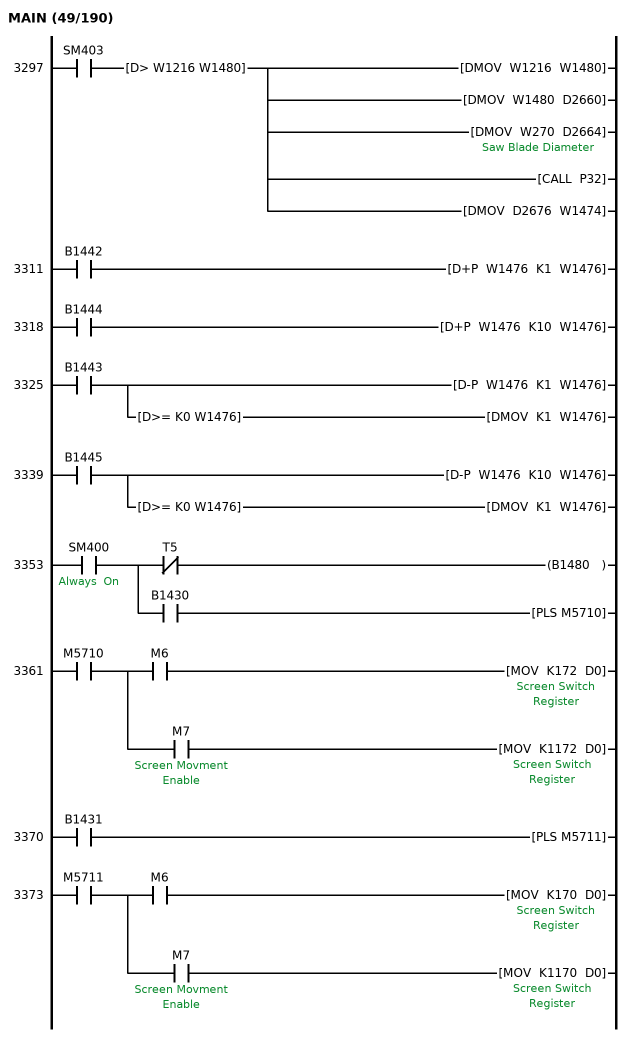
[picture p48: ladder of MAIN, rungs at steps 3297 to 3373]
3297  LD      SM403
      ANDD>   W1216 W1480
      DMOV    W1216 W1480
      DMOV    W1480 D2660
      DMOV    W270 D2664
      CALL    P32
      DMOV    D2676 W1474
3311  LD      B1442
      D+P     W1476 K1 W1476
3318  LD      B1444
      D+P     W1476 K10 W1476
3325  LD      B1443
      D-P     W1476 K1 W1476
      ANDD>=  K0 W1476
      DMOV    K1 W1476
3339  LD      B1445
      D-P     W1476 K10 W1476
      ANDD>=  K0 W1476
      DMOV    K1 W1476
3353  LD      SM400  ; Always  On
      MPS
      ANI     T5
      OUT     B1480
      MPP
      AND     B1430
      PLS     M5710
3361  LD      M5710
      MPS
      AND     M6
      MOV     K172 D0
      MPP
      AND     M7  ; Screen Movment Enable
      MOV     K1172 D0
3370  LD      B1431
      PLS     M5711
3373  LD      M5711
      MPS
      AND     M6
      MOV     K170 D0
      MPP
      AND     M7  ; Screen Movment Enable
      MOV     K1170 D0
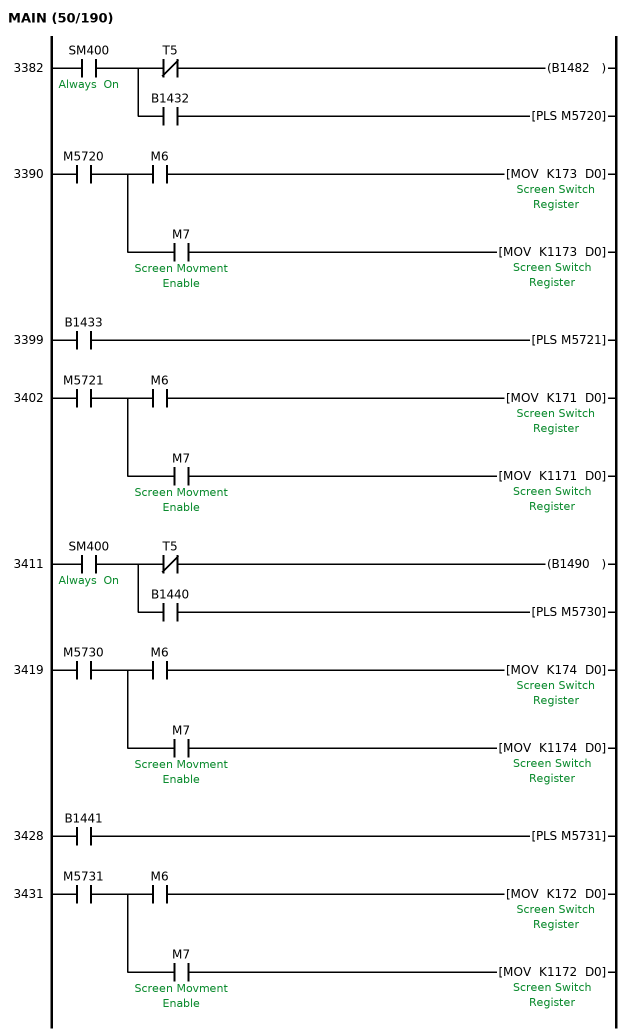
3382  LD      SM400  ; Always  On
      MPS
      ANI     T5
      OUT     B1482
      MPP
      AND     B1432
      PLS     M5720
3390  LD      M5720
      MPS
      AND     M6
      MOV     K173 D0
      MPP
      AND     M7  ; Screen Movment Enable
      MOV     K1173 D0
3399  LD      B1433
      PLS     M5721
3402  LD      M5721
      MPS
      AND     M6
      MOV     K171 D0
      MPP
      AND     M7  ; Screen Movment Enable
      MOV     K1171 D0
3411  LD      SM400  ; Always  On
      MPS
      ANI     T5
      OUT     B1490
      MPP
      AND     B1440
      PLS     M5730
3419  LD      M5730
      MPS
      AND     M6
      MOV     K174 D0
      MPP
      AND     M7  ; Screen Movment Enable
      MOV     K1174 D0
3428  LD      B1441
      PLS     M5731
3431  LD      M5731
      MPS
      AND     M6
      MOV     K172 D0
      MPP
      AND     M7  ; Screen Movment Enable
      MOV     K1172 D0
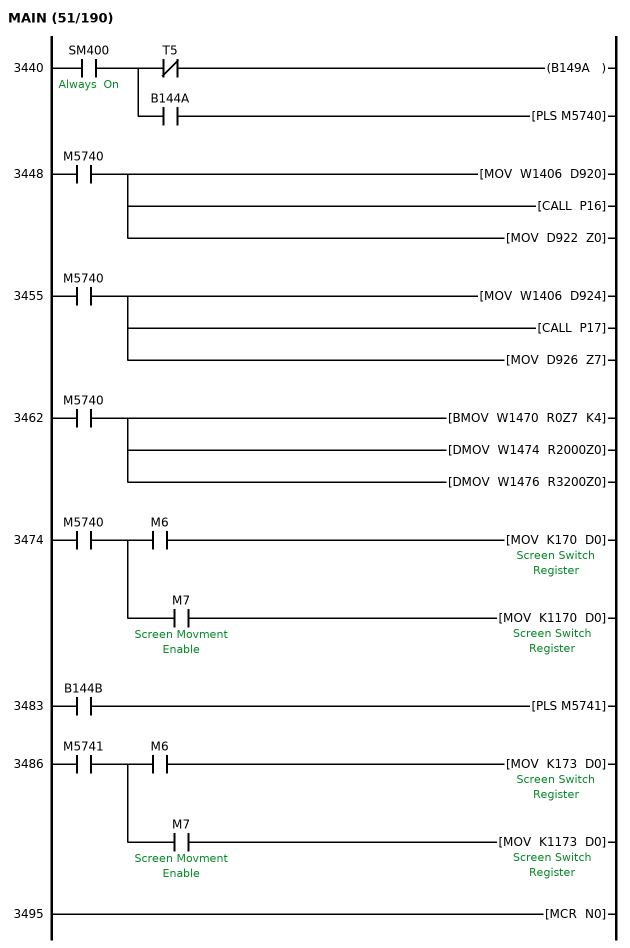
3440  LD      SM400  ; Always  On
      MPS
      ANI     T5
      OUT     B149A
      MPP
      AND     B144A
      PLS     M5740
3448  LD      M5740
      MOV     W1406 D920
      CALL    P16
      MOV     D922 Z0
3455  LD      M5740
      MOV     W1406 D924
      CALL    P17
      MOV     D926 Z7
3462  LD      M5740
      BMOV    W1470 R0Z7 K4
      DMOV    W1474 R2000Z0
      DMOV    W1476 R3200Z0
3474  LD      M5740
      MPS
      AND     M6
      MOV     K170 D0
      MPP
      AND     M7  ; Screen Movment Enable
      MOV     K1170 D0
3483  LD      B144B
      PLS     M5741
3486  LD      M5741
      MPS
      AND     M6
      MOV     K173 D0
      MPP
      AND     M7  ; Screen Movment Enable
      MOV     K1173 D0
3495  MCR     N0
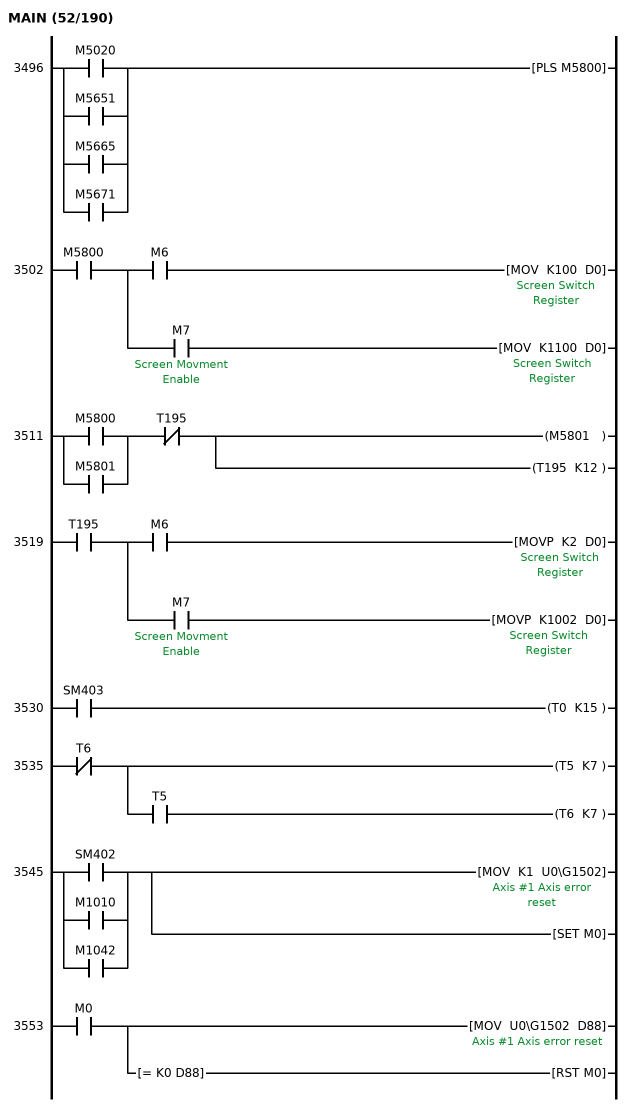
3496  LD      M5020
      OR      M5651
      OR      M5665
      OR      M5671
      PLS     M5800
3502  LD      M5800
      MPS
      AND     M6
      MOV     K100 D0
      MPP
      AND     M7  ; Screen Movment Enable
      MOV     K1100 D0
3511  LD      M5800
      OR      M5801
      ANI     T195
      OUT     M5801
      OUT     T195 K12
3519  LD      T195
      MPS
      AND     M6
      MOVP    K2 D0
      MPP
      AND     M7  ; Screen Movment Enable
      MOVP    K1002 D0
3530  LD      SM403
      OUT     T0 K15
3535  LDI     T6
      OUT     T5 K7
      AND     T5
      OUT     T6 K7
3545  LD      SM402
      OR      M1010
      OR      M1042
      MOV     K1 U0\G1502  ; Axis #1 Axis error reset
      SET     M0
3553  LD      M0
      MOV     U0\G1502 D88
      AND=    K0 D88
      RST     M0
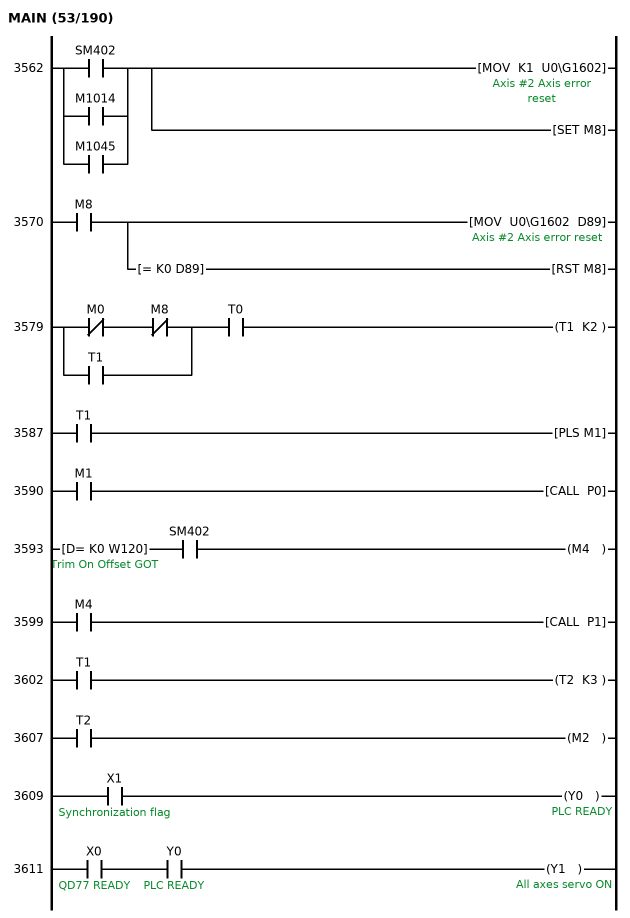
3562  LD      SM402
      OR      M1014
      OR      M1045
      MOV     K1 U0\G1602  ; Axis #2 Axis error reset
      SET     M8
3570  LD      M8
      MOV     U0\G1602 D89
      AND=    K0 D89
      RST     M8
3579  LDI     M0
      ANI     M8
      OR      T1
      AND     T0
      OUT     T1 K2
3587  LD      T1
      PLS     M1
3590  LD      M1
      CALL    P0
3593  LDD=    K0 W120  ; Trim On Offset GOT
      AND     SM402
      OUT     M4
3599  LD      M4
      CALL    P1
3602  LD      T1
      OUT     T2 K3
3607  LD      T2
      OUT     M2
3609  LD      X1  ; Synchronization flag
      OUT     Y0  ; PLC READY
3611  LD      X0  ; QD77 READY
      AND     Y0  ; PLC READY
      OUT     Y1  ; All axes servo ON
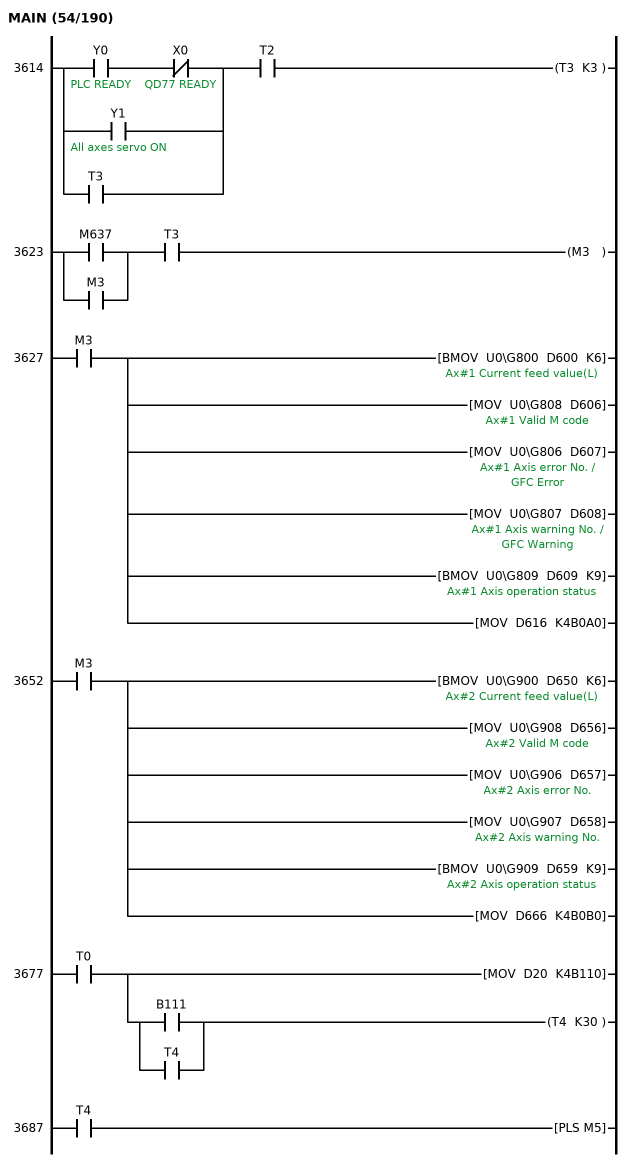
3614  LD      Y0  ; PLC READY
      ANI     X0  ; QD77 READY
      OR      Y1  ; All axes servo ON
      OR      T3
      AND     T2
      OUT     T3 K3
3623  LD      M637
      OR      M3
      AND     T3
      OUT     M3
3627  LD      M3
      BMOV    U0\G800 D600 K6  ; Ax#1 Current feed value(L)
      MOV     U0\G808 D606  ; Ax#1 Valid M code
      MOV     U0\G806 D607  ; Ax#1 Axis error No. / GFC Error
      MOV     U0\G807 D608  ; Ax#1 Axis warning No. / GFC Warning
      BMOV    U0\G809 D609 K9  ; Ax#1 Axis operation status
      MOV     D616 K4B0A0
3652  LD      M3
      BMOV    U0\G900 D650 K6  ; Ax#2 Current feed value(L)
      MOV     U0\G908 D656  ; Ax#2 Valid M code
      MOV     U0\G906 D657  ; Ax#2 Axis error No.
      MOV     U0\G907 D658  ; Ax#2 Axis warning No.
      BMOV    U0\G909 D659 K9  ; Ax#2 Axis operation status
      MOV     D666 K4B0B0
3677  LD      T0
      MOV     D20 K4B110
      LD      B111
      OR      T4
      ANB
      OUT     T4 K30
3687  LD      T4
      PLS     M5
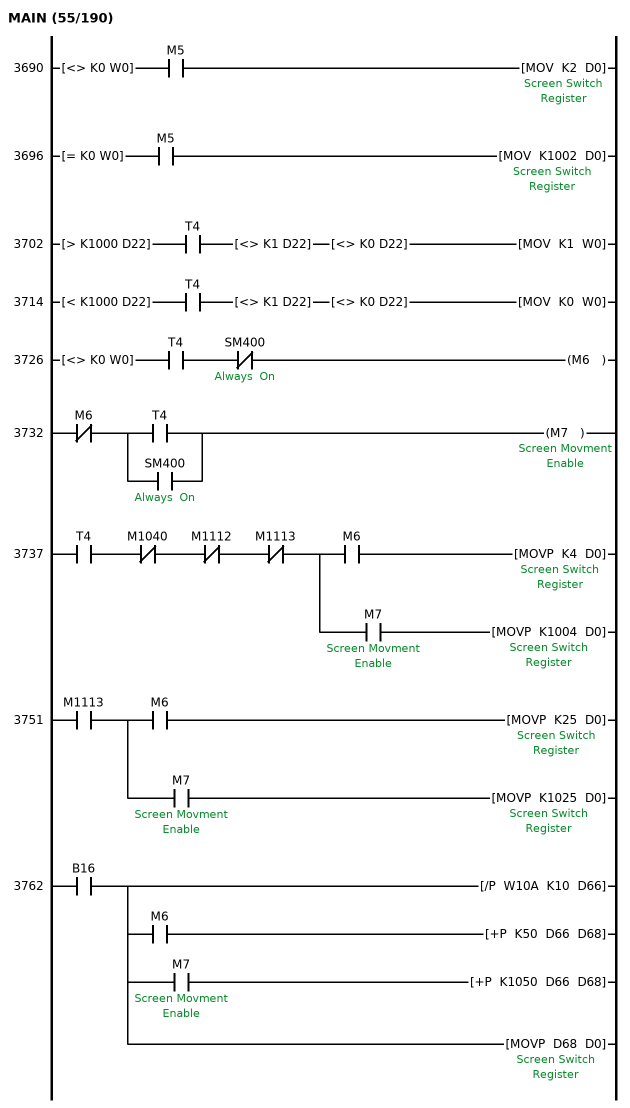
3690  LD<>    K0 W0
      AND     M5
      MOV     K2 D0
3696  LD=     K0 W0
      AND     M5
      MOV     K1002 D0
3702  LD>     K1000 D22
      AND     T4
      AND<>   K1 D22
      AND<>   K0 D22
      MOV     K1 W0
3714  LD<     K1000 D22
      AND     T4
      AND<>   K1 D22
      AND<>   K0 D22
      MOV     K0 W0
3726  LD<>    K0 W0
      AND     T4
      ANI     SM400  ; Always  On
      OUT     M6
3732  LDI     M6
      LD      T4
      OR      SM400  ; Always  On
      ANB
      OUT     M7  ; Screen Movment Enable
3737  LD      T4
      ANI     M1040
      ANI     M1112
      ANI     M1113
      MPS
      AND     M6
      MOVP    K4 D0
      MPP
      AND     M7  ; Screen Movment Enable
      MOVP    K1004 D0
3751  LD      M1113
      MPS
      AND     M6
      MOVP    K25 D0
      MPP
      AND     M7  ; Screen Movment Enable
      MOVP    K1025 D0
3762  LD      B16
      /P      W10A K10 D66
      MPS
      AND     M6
      +P      K50 D66 D68
      MRD
      AND     M7  ; Screen Movment Enable
      +P      K1050 D66 D68
      MPP
      MOVP    D68 D0
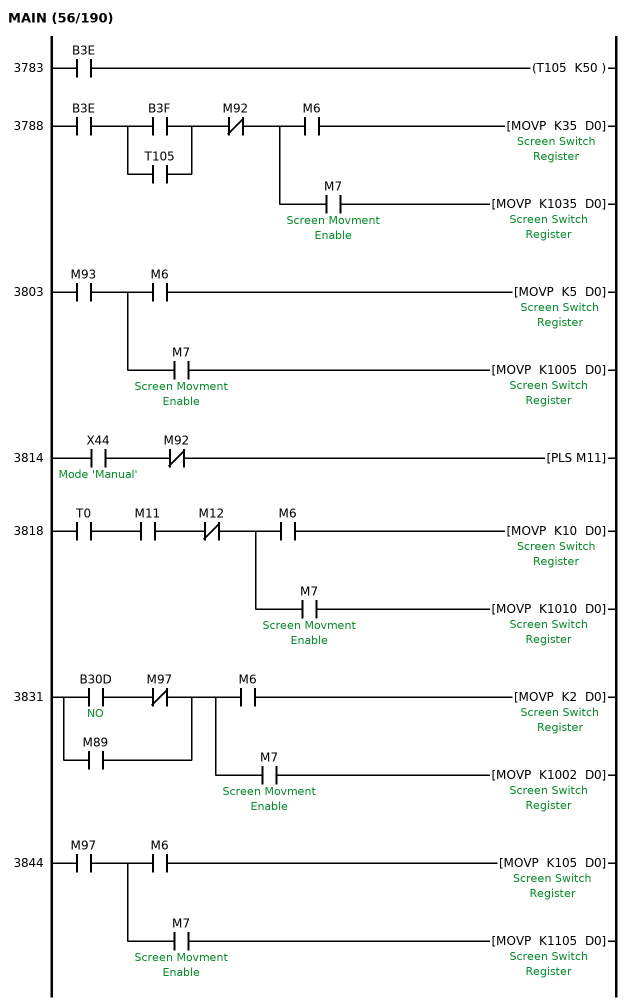
3783  LD      B3E
      OUT     T105 K50
3788  LD      B3E
      LD      B3F
      OR      T105
      ANB
      ANI     M92
      MPS
      AND     M6
      MOVP    K35 D0
      MPP
      AND     M7  ; Screen Movment Enable
      MOVP    K1035 D0
3803  LD      M93
      MPS
      AND     M6
      MOVP    K5 D0
      MPP
      AND     M7  ; Screen Movment Enable
      MOVP    K1005 D0
3814  LD      X44  ; Mode 'Manual'
      ANI     M92
      PLS     M11
3818  LD      T0
      AND     M11
      ANI     M12
      MPS
      AND     M6
      MOVP    K10 D0
      MPP
      AND     M7  ; Screen Movment Enable
      MOVP    K1010 D0
3831  LD      B30D  ; NO
      ANI     M97
      OR      M89
      MPS
      AND     M6
      MOVP    K2 D0
      MPP
      AND     M7  ; Screen Movment Enable
      MOVP    K1002 D0
3844  LD      M97
      MPS
      AND     M6
      MOVP    K105 D0
      MPP
      AND     M7  ; Screen Movment Enable
      MOVP    K1105 D0
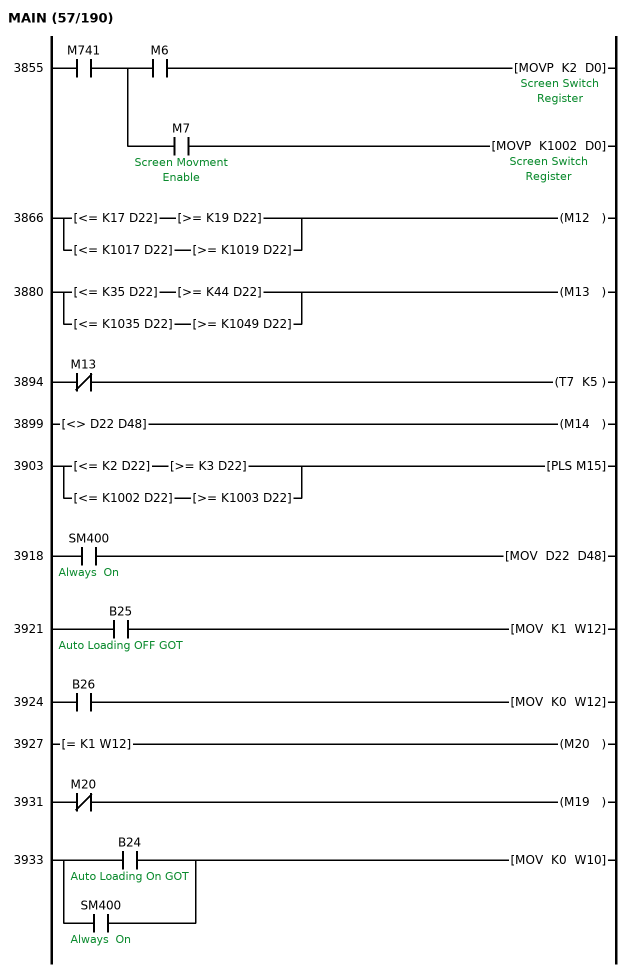
3855  LD      M741
      MPS
      AND     M6
      MOVP    K2 D0
      MPP
      AND     M7  ; Screen Movment Enable
      MOVP    K1002 D0
3866  LD<=    K17 D22
      AND>=   K19 D22
      LD<=    K1017 D22
      AND>=   K1019 D22
      ORB
      OUT     M12
3880  LD<=    K35 D22
      AND>=   K44 D22
      LD<=    K1035 D22
      AND>=   K1049 D22
      ORB
      OUT     M13
3894  LDI     M13
      OUT     T7 K5
3899  LD<>    D22 D48
      OUT     M14
3903  LD<=    K2 D22
      AND>=   K3 D22
      LD<=    K1002 D22
      AND>=   K1003 D22
      ORB
      PLS     M15
3918  LD      SM400  ; Always  On
      MOV     D22 D48
3921  LD      B25  ; Auto Loading OFF GOT
      MOV     K1 W12
3924  LD      B26
      MOV     K0 W12
3927  LD=     K1 W12
      OUT     M20
3931  LDI     M20
      OUT     M19
3933  LD      B24  ; Auto Loading On GOT
      OR      SM400  ; Always  On
      MOV     K0 W10
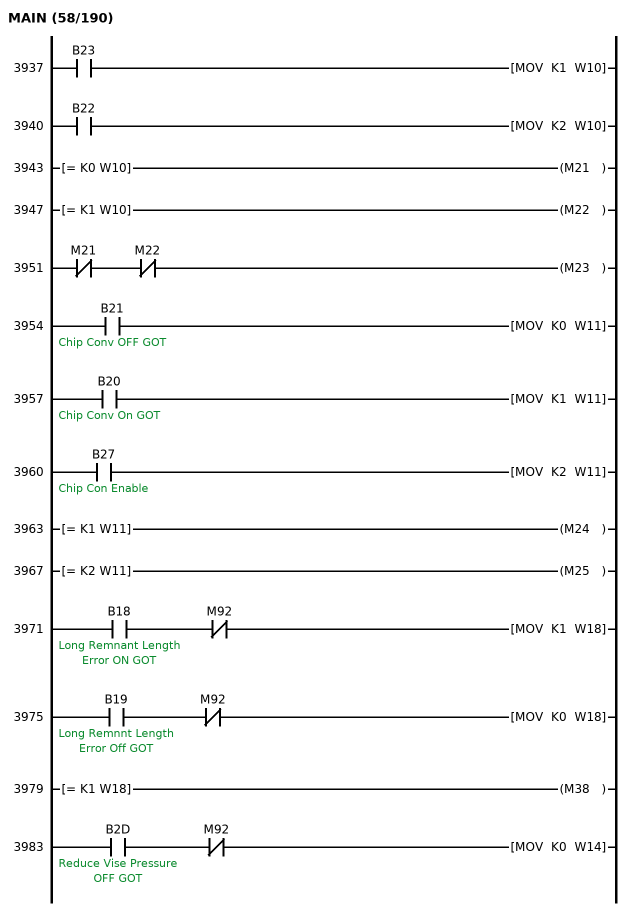
3937  LD      B23
      MOV     K1 W10
3940  LD      B22
      MOV     K2 W10
3943  LD=     K0 W10
      OUT     M21
3947  LD=     K1 W10
      OUT     M22
3951  LDI     M21
      ANI     M22
      OUT     M23
3954  LD      B21  ; Chip Conv OFF GOT
      MOV     K0 W11
3957  LD      B20  ; Chip Conv On GOT
      MOV     K1 W11
3960  LD      B27  ; Chip Con Enable
      MOV     K2 W11
3963  LD=     K1 W11
      OUT     M24
3967  LD=     K2 W11
      OUT     M25
3971  LD      B18  ; Long Remnant Length Error ON GOT
      ANI     M92
      MOV     K1 W18
3975  LD      B19  ; Long Remnnt Length Error Off GOT
      ANI     M92
      MOV     K0 W18
3979  LD=     K1 W18
      OUT     M38
3983  LD      B2D  ; Reduce Vise Pressure OFF GOT
      ANI     M92
      MOV     K0 W14
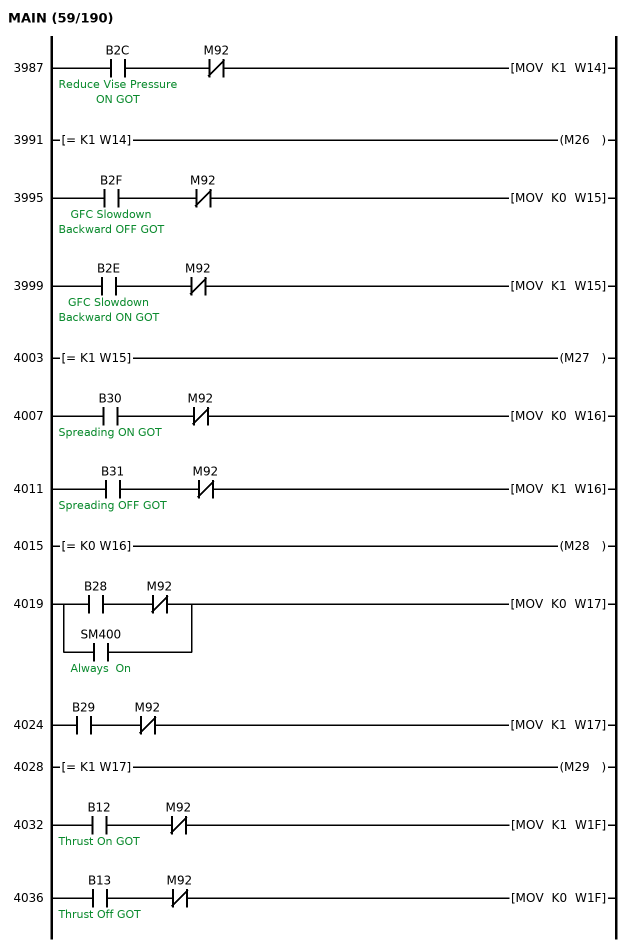
3987  LD      B2C  ; Reduce Vise Pressure ON GOT
      ANI     M92
      MOV     K1 W14
3991  LD=     K1 W14
      OUT     M26
3995  LD      B2F  ; GFC Slowdown Backward OFF GOT
      ANI     M92
      MOV     K0 W15
3999  LD      B2E  ; GFC Slowdown Backward ON GOT
      ANI     M92
      MOV     K1 W15
4003  LD=     K1 W15
      OUT     M27
4007  LD      B30  ; Spreading ON GOT
      ANI     M92
      MOV     K0 W16
4011  LD      B31  ; Spreading OFF GOT
      ANI     M92
      MOV     K1 W16
4015  LD=     K0 W16
      OUT     M28
4019  LD      B28
      ANI     M92
      OR      SM400  ; Always  On
      MOV     K0 W17
4024  LD      B29
      ANI     M92
      MOV     K1 W17
4028  LD=     K1 W17
      OUT     M29
4032  LD      B12  ; Thrust On GOT
      ANI     M92
      MOV     K1 W1F
4036  LD      B13  ; Thrust Off GOT
      ANI     M92
      MOV     K0 W1F
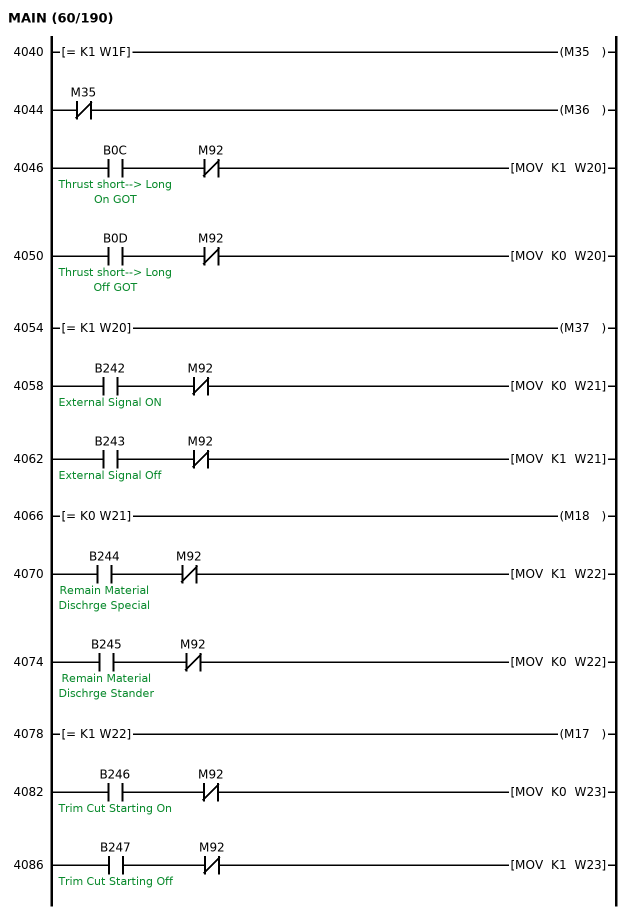
4040  LD=     K1 W1F
      OUT     M35
4044  LDI     M35
      OUT     M36
4046  LD      B0C  ; Thrust short--> Long On GOT
      ANI     M92
      MOV     K1 W20
4050  LD      B0D  ; Thrust short--> Long Off GOT
      ANI     M92
      MOV     K0 W20
4054  LD=     K1 W20
      OUT     M37
4058  LD      B242  ; External Signal ON
      ANI     M92
      MOV     K0 W21
4062  LD      B243  ; External Signal Off
      ANI     M92
      MOV     K1 W21
4066  LD=     K0 W21
      OUT     M18
4070  LD      B244  ; Remain Material Dischrge Special
      ANI     M92
      MOV     K1 W22
4074  LD      B245  ; Remain Material Dischrge Stander
      ANI     M92
      MOV     K0 W22
4078  LD=     K1 W22
      OUT     M17
4082  LD      B246  ; Trim Cut Starting On
      ANI     M92
      MOV     K0 W23
4086  LD      B247  ; Trim Cut Starting Off
      ANI     M92
      MOV     K1 W23
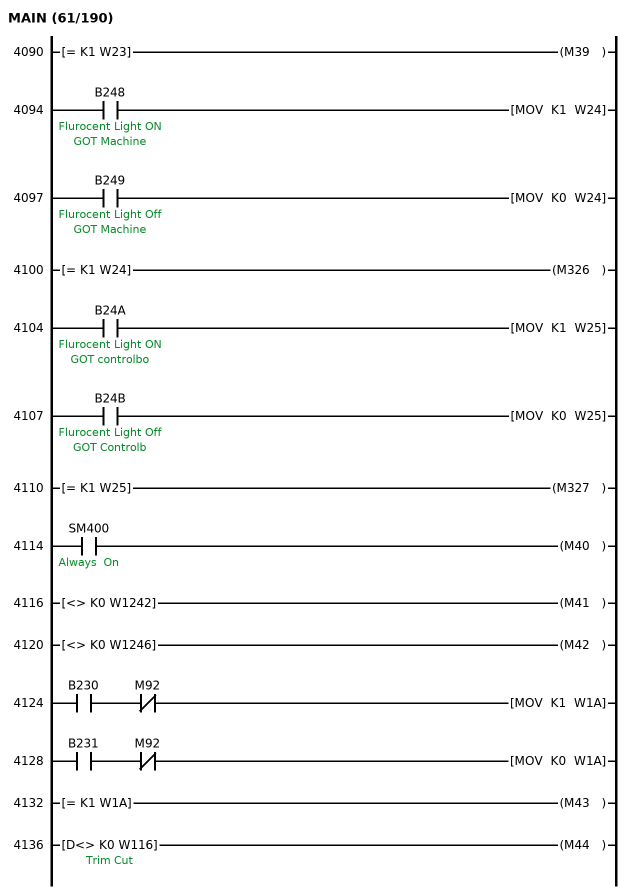
4090  LD=     K1 W23
      OUT     M39
4094  LD      B248  ; Flurocent Light ON GOT Machine
      MOV     K1 W24
4097  LD      B249  ; Flurocent Light Off GOT Machine
      MOV     K0 W24
4100  LD=     K1 W24
      OUT     M326
4104  LD      B24A  ; Flurocent Light ON GOT controlbo
      MOV     K1 W25
4107  LD      B24B  ; Flurocent Light Off GOT Controlb
      MOV     K0 W25
4110  LD=     K1 W25
      OUT     M327
4114  LD      SM400  ; Always  On
      OUT     M40
4116  LD<>    K0 W1242
      OUT     M41
4120  LD<>    K0 W1246
      OUT     M42
4124  LD      B230
      ANI     M92
      MOV     K1 W1A
4128  LD      B231
      ANI     M92
      MOV     K0 W1A
4132  LD=     K1 W1A
      OUT     M43
4136  LDD<>   K0 W116  ; Trim Cut
      OUT     M44
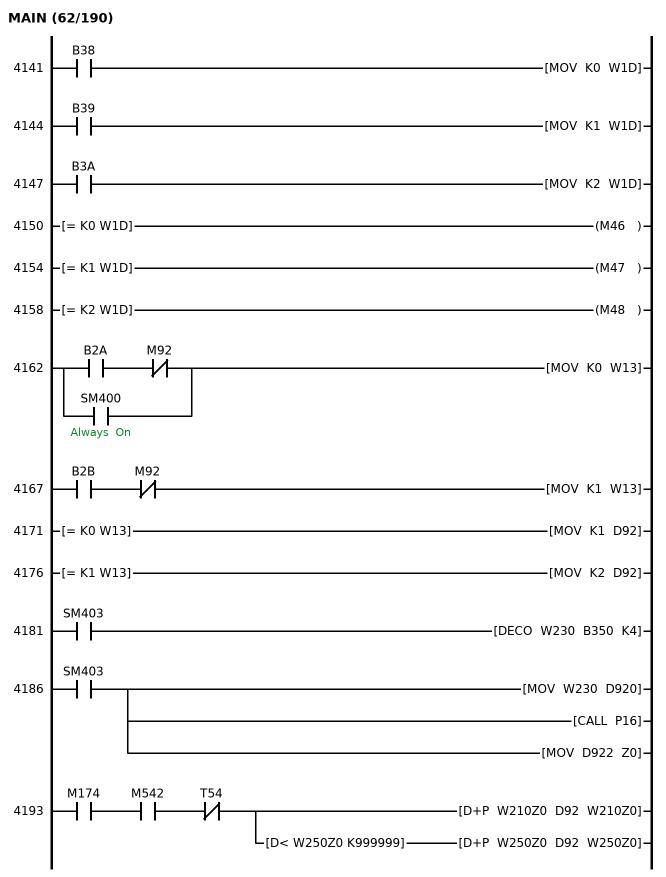
4141  LD      B38
      MOV     K0 W1D
4144  LD      B39
      MOV     K1 W1D
4147  LD      B3A
      MOV     K2 W1D
4150  LD=     K0 W1D
      OUT     M46
4154  LD=     K1 W1D
      OUT     M47
4158  LD=     K2 W1D
      OUT     M48
4162  LD      B2A
      ANI     M92
      OR      SM400  ; Always  On
      MOV     K0 W13
4167  LD      B2B
      ANI     M92
      MOV     K1 W13
4171  LD=     K0 W13
      MOV     K1 D92
4176  LD=     K1 W13
      MOV     K2 D92
4181  LD      SM403
      DECO    W230 B350 K4
4186  LD      SM403
      MOV     W230 D920
      CALL    P16
      MOV     D922 Z0
4193  LD      M174
      AND     M542
      ANI     T54
      D+P     W210Z0 D92 W210Z0
      ANDD<   W250Z0 K999999
      D+P     W250Z0 D92 W250Z0
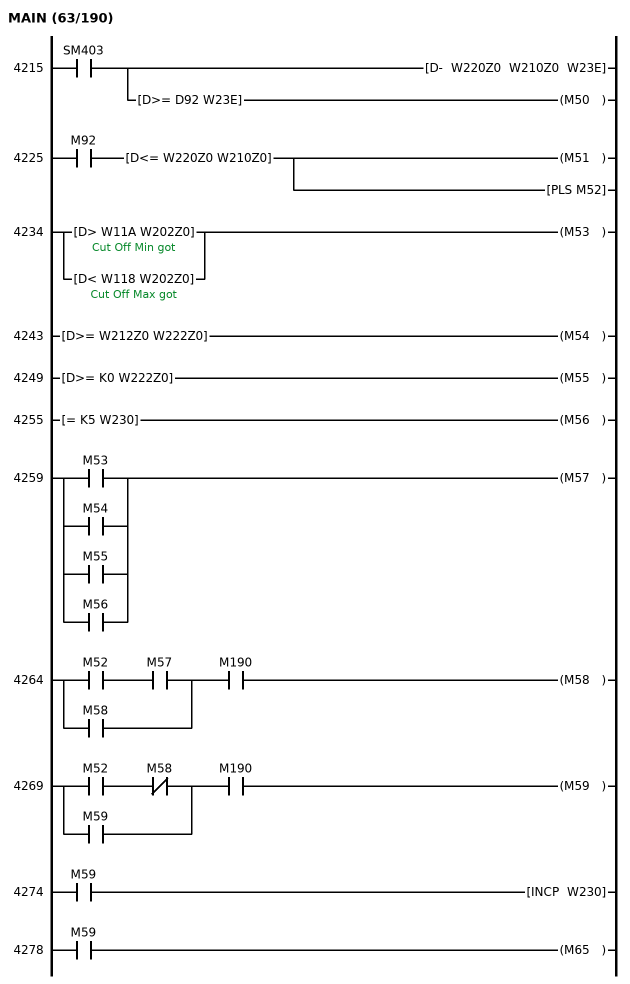
4215  LD      SM403
      D-      W220Z0 W210Z0 W23E
      ANDD>=  D92 W23E
      OUT     M50
4225  LD      M92
      ANDD<=  W220Z0 W210Z0
      OUT     M51
      PLS     M52
4234  LDD>    W11A W202Z0  ; Cut Off Min got
      ORD<    W118 W202Z0  ; Cut Off Max got
      OUT     M53
4243  LDD>=   W212Z0 W222Z0
      OUT     M54
4249  LDD>=   K0 W222Z0
      OUT     M55
4255  LD=     K5 W230
      OUT     M56
4259  LD      M53
      OR      M54
      OR      M55
      OR      M56
      OUT     M57
4264  LD      M52
      AND     M57
      OR      M58
      AND     M190
      OUT     M58
4269  LD      M52
      ANI     M58
      OR      M59
      AND     M190
      OUT     M59
4274  LD      M59
      INCP    W230
4278  LD      M59
      OUT     M65
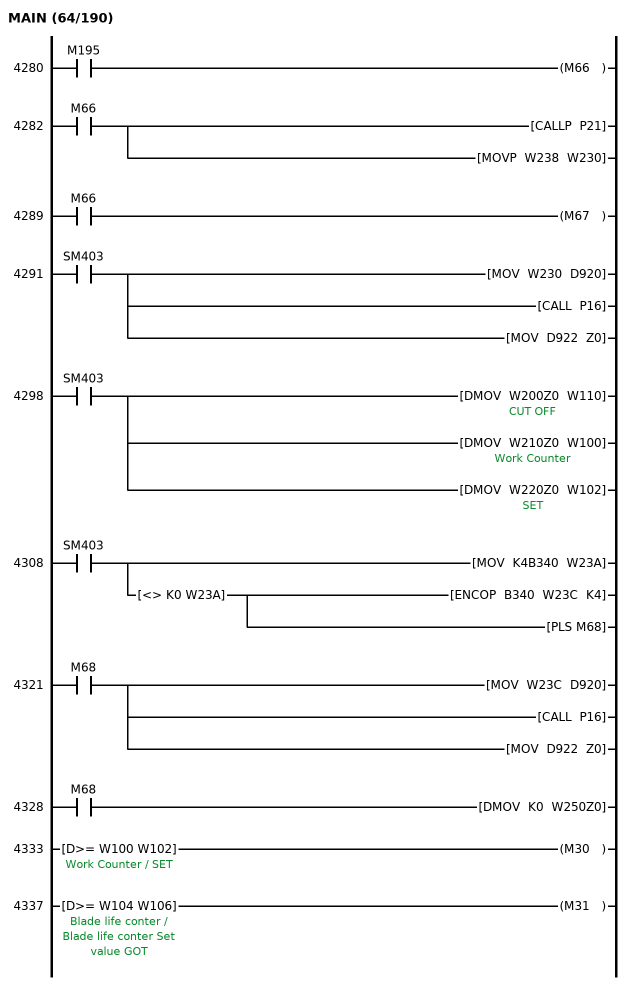
4280  LD      M195
      OUT     M66
4282  LD      M66
      CALLP   P21
      MOVP    W238 W230
4289  LD      M66
      OUT     M67
4291  LD      SM403
      MOV     W230 D920
      CALL    P16
      MOV     D922 Z0
4298  LD      SM403
      DMOV    W200Z0 W110  ; CUT OFF
      DMOV    W210Z0 W100  ; Work Counter
      DMOV    W220Z0 W102  ; SET
4308  LD      SM403
      MOV     K4B340 W23A
      AND<>   K0 W23A
      ENCOP   B340 W23C K4
      PLS     M68
4321  LD      M68
      MOV     W23C D920
      CALL    P16
      MOV     D922 Z0
4328  LD      M68
      DMOV    K0 W250Z0
4333  LDD>=   W100 W102  ; Work Counter / SET
      OUT     M30
4337  LDD>=   W104 W106  ; Blade life conter / Blade life conter Set value GOT
      OUT     M31
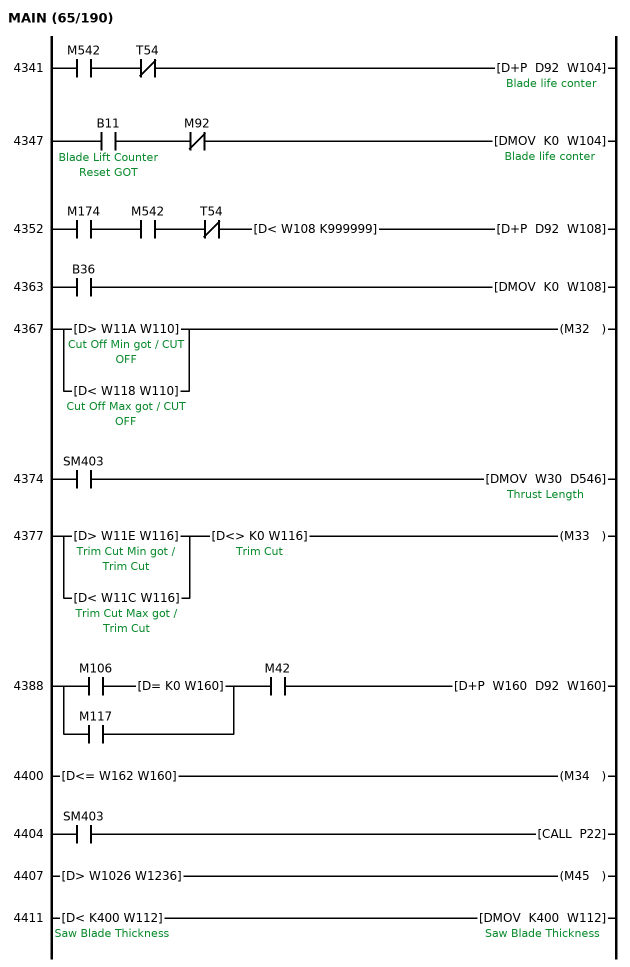
4341  LD      M542
      ANI     T54
      D+P     D92 W104
4347  LD      B11  ; Blade Lift Counter Reset GOT
      ANI     M92
      DMOV    K0 W104
4352  LD      M174
      AND     M542
      ANI     T54
      ANDD<   W108 K999999
      D+P     D92 W108
4363  LD      B36
      DMOV    K0 W108
4367  LDD>    W11A W110  ; Cut Off Min got / CUT OFF
      ORD<    W118 W110  ; Cut Off Max got / CUT OFF
      OUT     M32
4374  LD      SM403
      DMOV    W30 D546  ; Thrust Length
4377  LDD>    W11E W116  ; Trim Cut Min got / Trim Cut
      ORD<    W11C W116  ; Trim Cut Max got / Trim Cut
      ANDD<>  K0 W116  ; Trim Cut
      OUT     M33
4388  LD      M106
      ANDD=   K0 W160
      OR      M117
      AND     M42
      D+P     W160 D92 W160
4400  LDD<=   W162 W160
      OUT     M34
4404  LD      SM403
      CALL    P22
4407  LDD>    W1026 W1236
      OUT     M45
4411  LDD<    K400 W112  ; Saw Blade Thickness
      DMOV    K400 W112
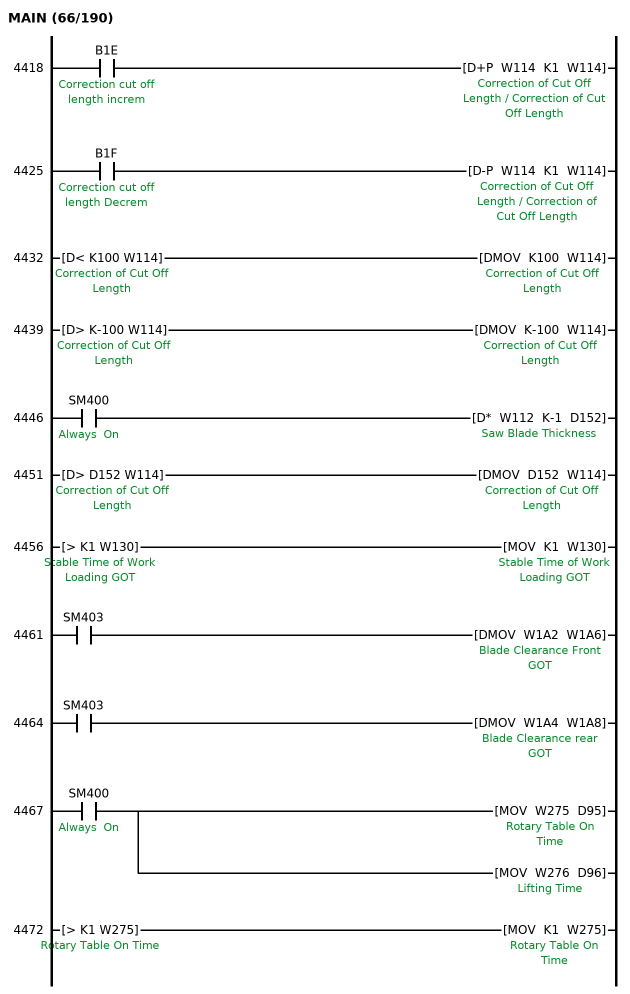
4418  LD      B1E  ; Correction cut off length increm
      D+P     W114 K1 W114  ; Correction of Cut Off Length
4425  LD      B1F  ; Correction cut off length Decrem
      D-P     W114 K1 W114
4432  LDD<    K100 W114  ; Correction of Cut Off Length
      DMOV    K100 W114
4439  LDD>    K-100 W114  ; Correction of Cut Off Length
      DMOV    K-100 W114
4446  LD      SM400  ; Always  On
      D*      W112 K-1 D152
4451  LDD>    D152 W114  ; Correction of Cut Off Length
      DMOV    D152 W114
4456  LD>     K1 W130  ; Stable Time of Work Loading GOT
      MOV     K1 W130
4461  LD      SM403
      DMOV    W1A2 W1A6  ; Blade Clearance Front GOT
4464  LD      SM403
      DMOV    W1A4 W1A8  ; Blade Clearance rear GOT
4467  LD      SM400  ; Always  On
      MOV     W275 D95  ; Rotary Table On Time
      MOV     W276 D96  ; Lifting Time
4472  LD>     K1 W275  ; Rotary Table On Time
      MOV     K1 W275
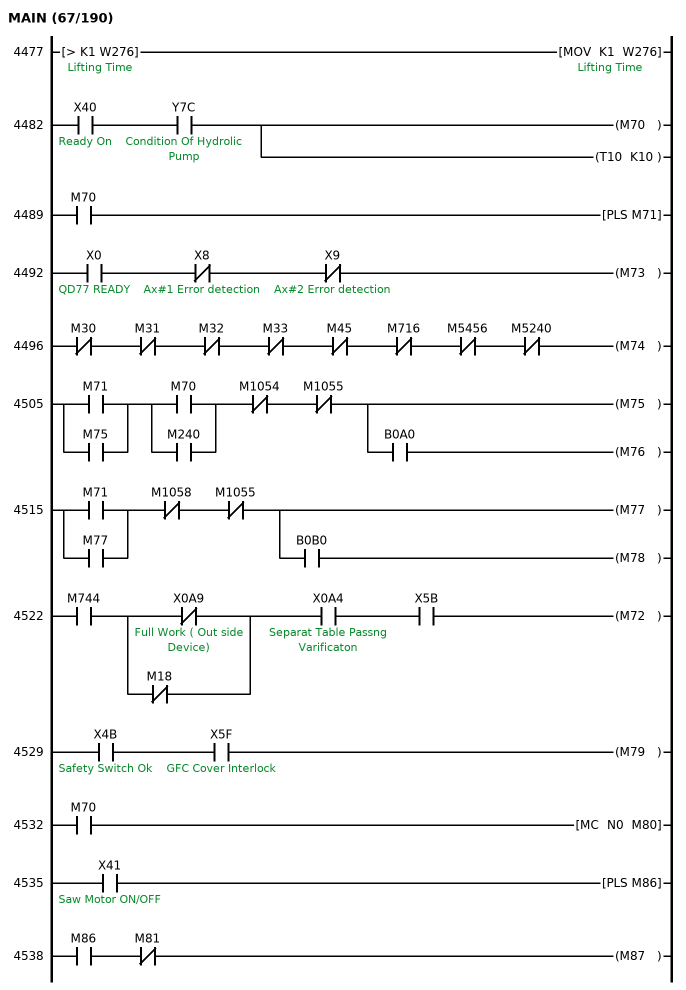
4477  LD>     K1 W276  ; Lifting Time
      MOV     K1 W276
4482  LD      X40  ; Ready On
      AND     Y7C  ; Condition Of Hydrolic Pump
      OUT     M70
      OUT     T10 K10
4489  LD      M70
      PLS     M71
4492  LD      X0  ; QD77 READY
      ANI     X8  ; Ax#1 Error detection
      ANI     X9  ; Ax#2 Error detection
      OUT     M73
4496  LDI     M30
      ANI     M31
      ANI     M32
      ANI     M33
      ANI     M45
      ANI     M716
      ANI     M5456
      ANI     M5240
      OUT     M74
4505  LD      M71
      OR      M75
      LD      M70
      OR      M240
      ANB
      ANI     M1054
      ANI     M1055
      OUT     M75
      AND     B0A0
      OUT     M76
4515  LD      M71
      OR      M77
      ANI     M1058
      ANI     M1055
      OUT     M77
      AND     B0B0
      OUT     M78
4522  LD      M744
      LDI     X0A9  ; Full Work ( Out side Device)
      ORI     M18
      ANB
      AND     X0A4  ; Separat Table Passng Varificaton
      AND     X5B
      OUT     M72
4529  LD      X4B  ; Safety Switch Ok
      AND     X5F  ; GFC Cover Interlock
      OUT     M79
4532  LD      M70
      MC      N0 M80
4535  LD      X41  ; Saw Motor ON/OFF
      PLS     M86
4538  LD      M86
      ANI     M81
      OUT     M87
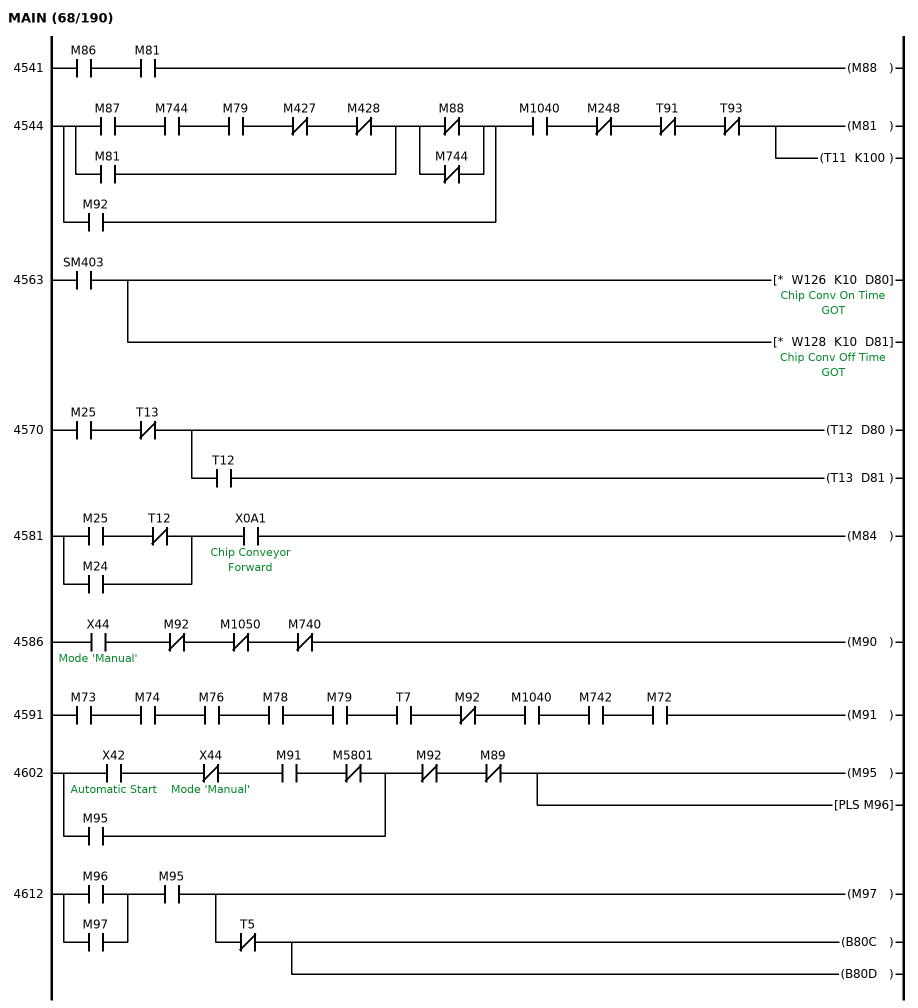
4541  LD      M86
      AND     M81
      OUT     M88
4544  LD      M87
      AND     M744
      AND     M79
      ANI     M427
      ANI     M428
      OR      M81
      LDI     M88
      ORI     M744
      ANB
      OR      M92
      AND     M1040
      ANI     M248
      ANI     T91
      ANI     T93
      OUT     M81
      OUT     T11 K100
4563  LD      SM403
      *       W126 K10 D80  ; Chip Conv On Time GOT
      *       W128 K10 D81  ; Chip Conv Off Time GOT
4570  LD      M25
      ANI     T13
      OUT     T12 D80
      AND     T12
      OUT     T13 D81
4581  LD      M25
      ANI     T12
      OR      M24
      AND     X0A1  ; Chip Conveyor Forward
      OUT     M84
4586  LD      X44  ; Mode 'Manual'
      ANI     M92
      ANI     M1050
      ANI     M740
      OUT     M90
4591  LD      M73
      AND     M74
      AND     M76
      AND     M78
      AND     M79
      AND     T7
      ANI     M92
      AND     M1040
      AND     M742
      AND     M72
      OUT     M91
4602  LD      X42  ; Automatic Start
      ANI     X44  ; Mode 'Manual'
      AND     M91
      ANI     M5801
      OR      M95
      ANI     M92
      ANI     M89
      OUT     M95
      PLS     M96
4612  LD      M96
      OR      M97
      AND     M95
      OUT     M97
      ANI     T5
      OUT     B80C
      OUT     B80D
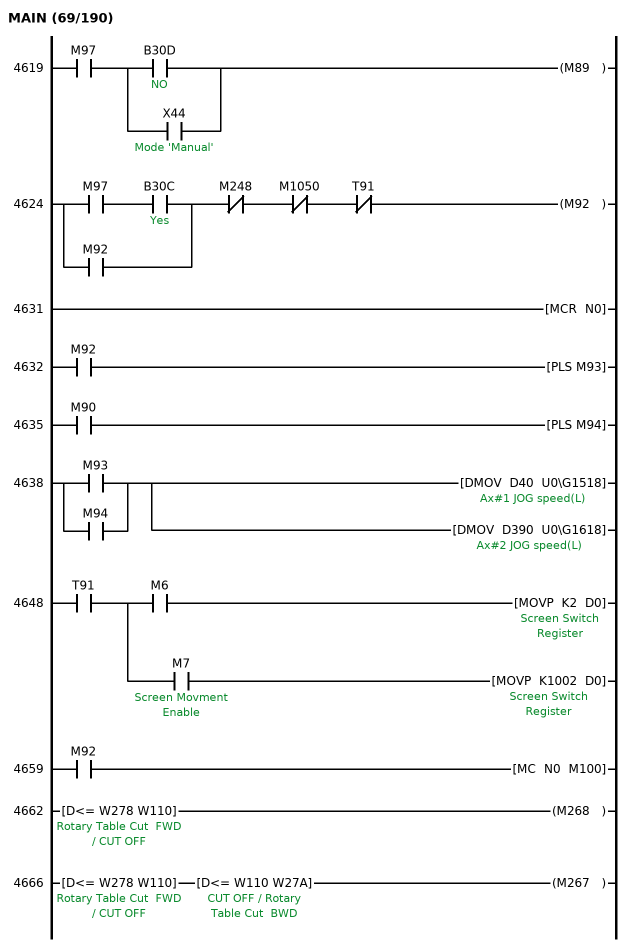
4619  LD      M97
      LD      B30D  ; NO
      OR      X44  ; Mode 'Manual'
      ANB
      OUT     M89
4624  LD      M97
      AND     B30C  ; Yes
      OR      M92
      ANI     M248
      ANI     M1050
      ANI     T91
      OUT     M92
4631  MCR     N0
4632  LD      M92
      PLS     M93
4635  LD      M90
      PLS     M94
4638  LD      M93
      OR      M94
      DMOV    D40 U0\G1518  ; Ax#1 JOG speed(L)
      DMOV    D390 U0\G1618  ; Ax#2 JOG speed(L)
4648  LD      T91
      MPS
      AND     M6
      MOVP    K2 D0
      MPP
      AND     M7  ; Screen Movment Enable
      MOVP    K1002 D0
4659  LD      M92
      MC      N0 M100
4662  LDD<=   W278 W110  ; Rotary Table Cut  FWD / CUT OFF
      OUT     M268
4666  LDD<=   W278 W110  ; Rotary Table Cut  FWD / CUT OFF
      ANDD<=  W110 W27A  ; CUT OFF / Rotary Table Cut  BWD
      OUT     M267
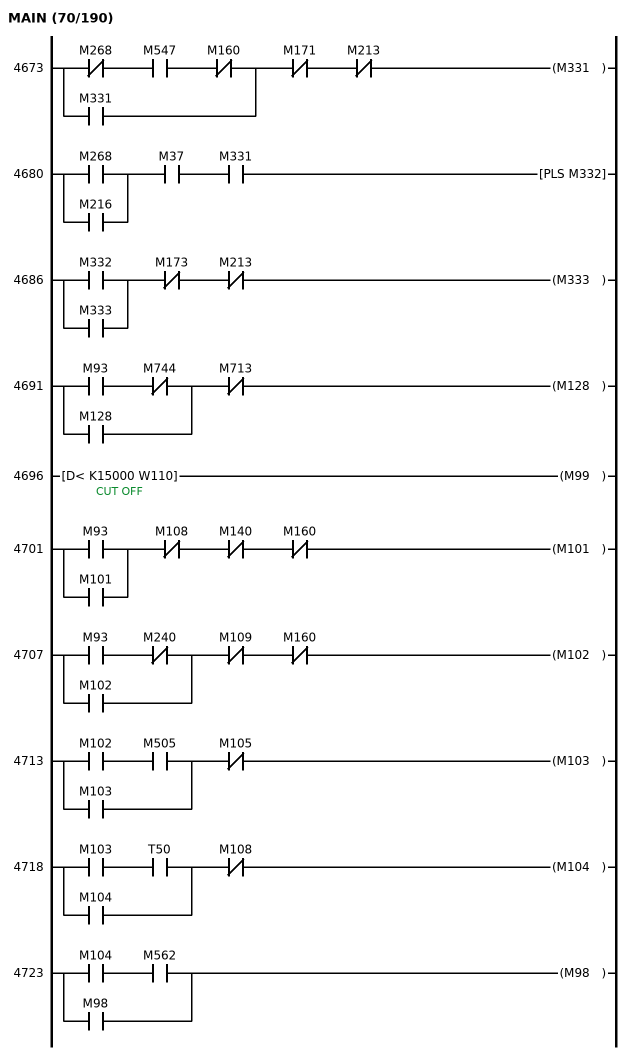
4673  LDI     M268
      AND     M547
      ANI     M160
      OR      M331
      ANI     M171
      ANI     M213
      OUT     M331
4680  LD      M268
      OR      M216
      AND     M37
      AND     M331
      PLS     M332
4686  LD      M332
      OR      M333
      ANI     M173
      ANI     M213
      OUT     M333
4691  LD      M93
      ANI     M744
      OR      M128
      ANI     M713
      OUT     M128
4696  LDD<    K15000 W110  ; CUT OFF
      OUT     M99
4701  LD      M93
      OR      M101
      ANI     M108
      ANI     M140
      ANI     M160
      OUT     M101
4707  LD      M93
      ANI     M240
      OR      M102
      ANI     M109
      ANI     M160
      OUT     M102
4713  LD      M102
      AND     M505
      OR      M103
      ANI     M105
      OUT     M103
4718  LD      M103
      AND     T50
      OR      M104
      ANI     M108
      OUT     M104
4723  LD      M104
      AND     M562
      OR      M98
      OUT     M98
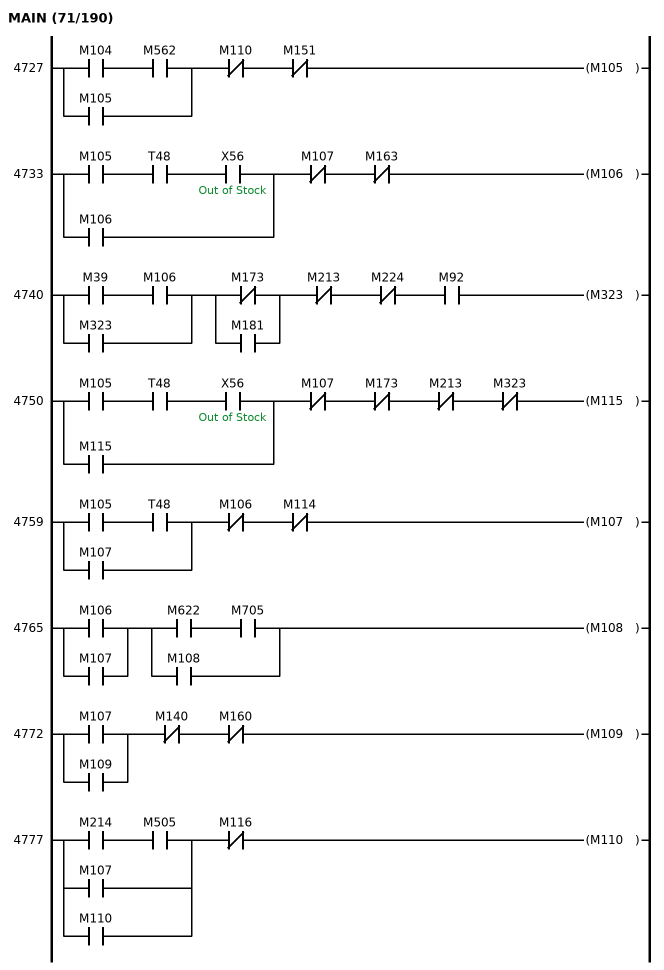
4727  LD      M104
      AND     M562
      OR      M105
      ANI     M110
      ANI     M151
      OUT     M105
4733  LD      M105
      AND     T48
      AND     X56  ; Out of Stock
      OR      M106
      ANI     M107
      ANI     M163
      OUT     M106
4740  LD      M39
      AND     M106
      OR      M323
      LDI     M173
      OR      M181
      ANB
      ANI     M213
      ANI     M224
      AND     M92
      OUT     M323
4750  LD      M105
      AND     T48
      AND     X56  ; Out of Stock
      OR      M115
      ANI     M107
      ANI     M173
      ANI     M213
      ANI     M323
      OUT     M115
4759  LD      M105
      AND     T48
      OR      M107
      ANI     M106
      ANI     M114
      OUT     M107
4765  LD      M106
      OR      M107
      LD      M622
      AND     M705
      OR      M108
      ANB
      OUT     M108
4772  LD      M107
      OR      M109
      ANI     M140
      ANI     M160
      OUT     M109
4777  LD      M214
      AND     M505
      OR      M107
      OR      M110
      ANI     M116
      OUT     M110
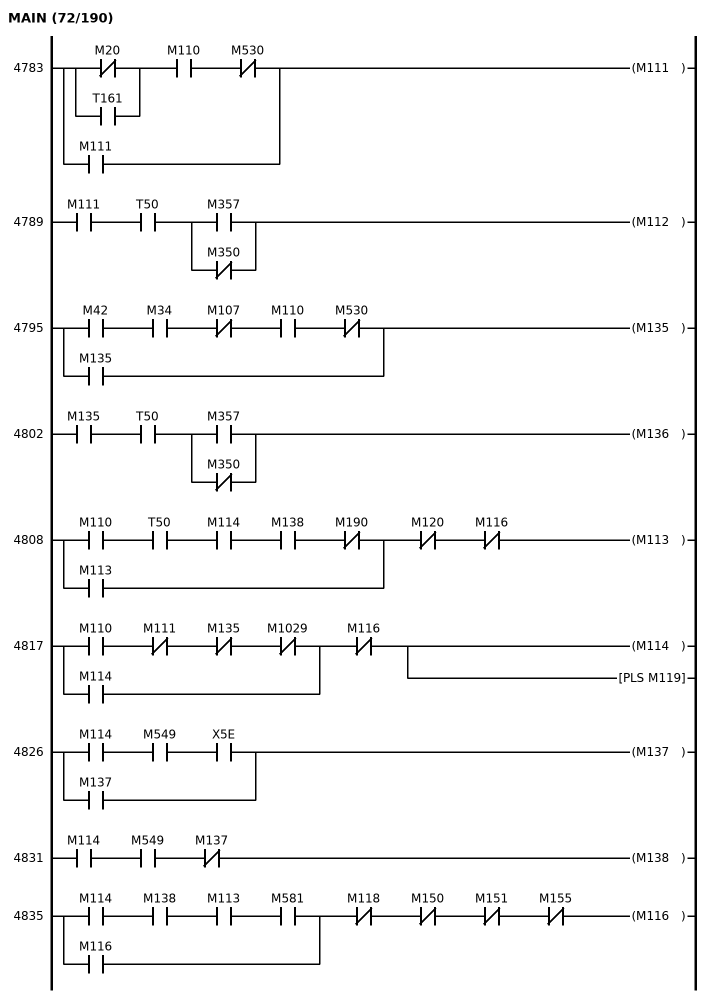
4783  LDI     M20
      OR      T161
      AND     M110
      ANI     M530
      OR      M111
      OUT     M111
4789  LD      M111
      AND     T50
      LD      M357
      ORI     M350
      ANB
      OUT     M112
4795  LD      M42
      AND     M34
      ANI     M107
      AND     M110
      ANI     M530
      OR      M135
      OUT     M135
4802  LD      M135
      AND     T50
      LD      M357
      ORI     M350
      ANB
      OUT     M136
4808  LD      M110
      AND     T50
      AND     M114
      AND     M138
      ANI     M190
      OR      M113
      ANI     M120
      ANI     M116
      OUT     M113
4817  LD      M110
      ANI     M111
      ANI     M135
      ANI     M1029
      OR      M114
      ANI     M116
      OUT     M114
      PLS     M119
4826  LD      M114
      AND     M549
      AND     X5E
      OR      M137
      OUT     M137
4831  LD      M114
      AND     M549
      ANI     M137
      OUT     M138
4835  LD      M114
      AND     M138
      AND     M113
      AND     M581
      OR      M116
      ANI     M118
      ANI     M150
      ANI     M151
      ANI     M155
      OUT     M116
